TYPE ST_ElementBaseEmulation :
(**************************************************************************************
 * 	Application		:	BoxControl Framework
 *	Revision		:	$Revision: 404529 $
 *	Revision date	:	$Date: 2018-04-23 08:21:38 +0200 (Mo., 23 Apr 2018) $
 *	Last changed by	:	$Author: b7bolm $
 *	URL				:	$URL: http://almscdc.swisslog.com/repo/SWPD/Development/BoxControlFramework/20_Release/trunk/01_Software/BCF/BCF/JumpStart/20_Product/11_Emu/13_Elements/10_Lib/10_Conv/01_DUTs/ST_ElementBaseEmulation.TcDUT $
 *
 *	Purpose			:	Function interface - Contains data which is provided by the
 *						function or is input from other objects.
 *
 * ------------------------------------------------------------------------------------
 *	Copyright Swisslog [IP AG], Switzerland. All rights reserved.
 * 
 * ------------------------------------------------------------------------------------
 *	
 * 	Revision History: 
 *
 * 	VERSION			DATE			INITIALS			DESCRIPTION
 *	0.1				01.01.2001		swl					Example
 *
 **************************************************************************************)
STRUCT
	rElementDataReal				: REFERENCE TO ST_ElementData; // Real Element data
	ElementDataEmpty				: ST_ElementData;
	rElementInterfaceReal			: REFERENCE TO ST_ElementInterface; // Real Element interface
	ElementInterfaceEmpty			: ST_ElementInterface;
	rSettingsElementReal			: REFERENCE TO ST_CFG_Element; // Settings of real element
	SettingsElementEmpty			: ST_CFG_Element;
	eMsgType						: E_ITC_MsgTypeConv;
	ERQ								: ST_ITC_ERQ;
END_STRUCT
END_TYPE

(* stored: Version 1.1.0.1, ProductVersion 3.1.4022.12
   DUT ST_ElementBaseEmulation: Id {a9eef1f9-0c6a-4933-8948-af698dbdf61c} *)
